// TIA Portal V17 export
// export: Created 2024-09-02T12:50:40.2321894Z, ExportSetting WithDefaults, DisplayName Totally Integrated Automation Portal, DisplayVersion V17, DisplayName TIA Portal Openness, DisplayVersion V17, DisplayName TIA Portal Version Control Interface, DisplayVersion V17, DisplayName STEP 7 Professional, DisplayVersion V17, DisplayName STEP 7 Safety, DisplayVersion V17, DisplayName WinCC Professional, DisplayVersion V17
TYPE "Scania_Variants"
// stored: IsFailsafeCompliant false
   STRUCT
      GR875 : Bool;
      GRS895 : Bool;
      GRSO895 : Bool;
      GR905 : Bool;
      GRS905 : Bool;
      GRSO905 : Bool;
      GRS925 : Bool;
      GRSO926 : Bool;
      GRSO935 : Bool;
      G16M : Bool;
      G25M : Bool;
      G25CM : Bool;
      G33M : Bool;
      G33CM : Bool;
      G38M : Bool;
      G38CM : Bool;
      G45CM : Bool;
   END_STRUCT;
END_TYPE
